FUNCTION F_Turbo_NC_NO_Valve_Logic : BOOL
VAR_INPUT
    i_stTurbo : ST_PTM; // Turbo Pump
    i_stISG : ST_VG; //Gauge measuring inlet Pressure e.g Pirani
    i_stBSG : ST_VG; //Gauge measureing backing pressure
    iq_stValve_NO : ST_VRC_NO; //Normally Open Valve directly sharing turbo pump vaccum volume.
    iq_stValve_NC : ST_VRC; //Normally Closed Valve directly sharing turbo pump vaccum volume.
    iq_stValve_NC_second :	ST_VRC; //Normally Open Valve on the other side of NO valve that also connects to roughing line.
    ads_Error_Present	:	BOOL; // ADS Communication: Watchdog and ADS Read Error Bit
    iq_stRoughRoughValve_NC: ST_VGC_2S; //Normally Closed Valve Downstream of iq_stValve_NC in Beamline Roughing Line.
    iq_stRoughRoughValve_NC_second: ST_VGC_2S; //Normally Closed Valve Downstream of iq_stValve_NC_second in Beamline Roughing Line.
    x_onBeamline :	BOOL; //Whether the  Turbopump/Endstation is mounted on the beamline or not.
END_VAR
VAR
END_VAR

IF (x_onBeamline) THEN
    F_Turbo_NC_NO_Valve_Logic := (i_stISG.xPRESS_OK AND i_stISG.rPRESS < i_stTurbo.rInletPressureSP) AND
                                    (i_stBSG.xPRESS_OK AND i_stBSG.rPRESS < i_stTurbo.rBackingPressureSP) AND
                                 ((iq_stValve_NC.i_xOpnLS AND iq_stRoughRoughValve_NC.eState = E_ValvePositionState.OPEN) OR
                                 (iq_stValve_NO.i_xOpnLS AND (iq_stValve_NC_second.i_xOpnLS AND
                                 iq_stRoughRoughValve_NC_second.eState = E_ValvePositionState.OPEN)))AND (NOT ads_Error_Present);
ELSE
    F_Turbo_NC_NO_Valve_Logic := (i_stISG.xPRESS_OK AND i_stISG.rPRESS < i_stTurbo.rInletPressureSP) AND
                           (i_stBSG.xPRESS_OK AND i_stBSG.rPRESS < i_stTurbo.rBackingPressureSP) AND
                            (iq_stValve_NC.i_xOpnLS OR(iq_stValve_NO.i_xOpnLS AND iq_stValve_NC_second.i_xOpnLS));
END_IF

END_FUNCTION

(* stored: Version 1.1.0.1, ProductVersion 3.1.4022.18
   POU F_Turbo_NC_NO_Valve_Logic: Id {08997993-57bb-47dd-af54-2b770ca6585d}, SpecialFunc None *)
